FUNCTION Det7 : LREAL
VAR_IN_OUT CONSTANT
	mat: Mat7d;
END_VAR
VAR
	dim : INT :=7;
	i,j,k:INT;
	m,n :INT;
	cofactorMat : Mat6d;
	matdet :matrix66_det;
	tmp :LREAL;
END_VAR

Det7:=0;
FOR i :=1 TO dim DO
	// get cofactor mat
	m:=1;
	n:=1;
	FOR j:=1 TO dim DO
		FOR k:=1 TO dim DO
			IF j<>1 AND k <> i THEN
				cofactorMat[m,n]:=mat[j,k];
				n:=n+1;
				IF n>=dim THEN
					m:=m+1;
					n:=1;
				END_IF
			END_IF
		END_FOR
	END_FOR
	
	Det7:=Det7+ mat[1,i]*EXPT(-1,1+i)*Det6(cofactorMat);
END_FOR

END_FUNCTION

(* stored: Version 1.1.0.1, ProductVersion 3.1.4024.12
   POU Det7: Id {a87caff6-9780-4148-8c5d-14158f678cc4}, SpecialFunc None *)
